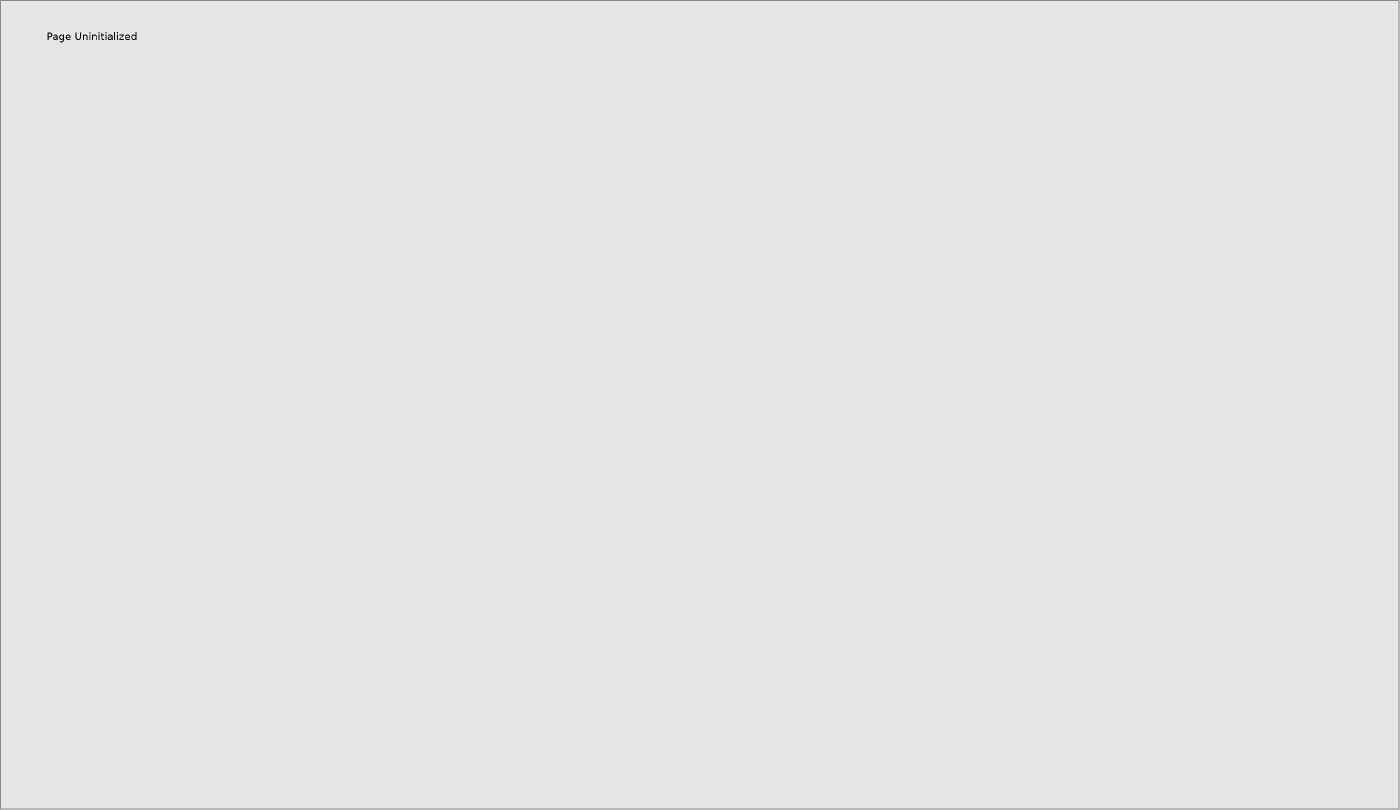
VISUALIZATION PageUninitialized  // 1520x880
    Label (25,25 150x30), "Page Uninitialized"
END_VISUALIZATION

(* stored: Version 1.1.0.1, ProductVersion 3.1.4024.9
   Visu PageUninitialized: Id {8065769f-ab69-4fc0-8d86-6905fea0168d} *)
